(* CoDeSys 2.3 export: FB_LAMP.EXP *)

(* POU FBs/FB_Lamp, ST *)
(*
 TODO: REACTION
*)
FUNCTION_BLOCK FB_Lamp
VAR_INPUT
	ON_OFF: BOOL;   (* on/off on pulse, ignored if FORCE = TRUE *)
	ON: BOOL;   (* on on pulse, ignored if FORCE = TRUE *)
	OFF: BOOL;   (* off on pulse, ignored if FORCE = TRUE *)
	PT: TIME := t#30s;   (* auto-off aka on-time; see also: expandPT *)
	OFF_BLOCK_ON: TIME := t#15s;   (* after off block ON for the time specified *)
	REACTION: TIME := t#600ms;   (* TODO: do not change state right after statechange *)
	FORCE: BOOL;   (* if true, force output on/off, depending on FORCE_ON;
			  during FORCE, IN is ignored
			  during FORCE, PT is expanded if Q = TRUE *)
	FORCE_ON: BOOL;   (* if false and FORCE, then force off *)
	ROOM: STRING;
	LOCATION: STRING;
END_VAR
VAR_OUTPUT RETAIN PERSISTENT
	usageTime: TIME := t#0ms;
	usageDays: UINT := 0;
	usageCounterSwitchOn: UDINT := 0;
END_VAR
VAR_OUTPUT
	Q: BOOL;   (* lamp on / off *)
END_VAR
VAR
	viText: STRING; (* ro by visualisation *)
	viOnTimer: TIME; (* ro by visualisation *)
	viOffTimer: TIME; (* ro by visualisation *)
	viOnOff: BOOL; (* wo by visualisation *)
	onTimer: TOF;
	offTimer: TOF;
	onTrigger: R_TRIG;
	onOffTrigger: R_TRIG;
	offTrigger: R_TRIG;
	forceOnTrigger: R_TRIG;
	forceOffTrigger: F_TRIG;
	forceOnTime: TIME;
	startOpTrigger: R_TRIG;
	stopOpTrigger: F_TRIG;
	opTimetracker: TIME;
	now: TIME;
	extendPT: TIME;   (* added to onTimer.PT *)
END_VAR
VAR CONSTANT
	MAX_TIME: TIME := T#71582m47s295ms;
END_VAR
viText := CONCAT(ROOM, '$N');
viText := CONCAT(viText, LOCATION);
(* viOnTimer and viOffTimer are set later *)

now := TIME();

forceOnTrigger(CLK := FORCE);
forceOffTrigger(CLK := FORCE);
IF forceOnTrigger.Q AND onTimer.Q THEN
	forceOnTime := now;
ELSIF forceOffTrigger.Q AND onTimer.Q THEN
	IF (now < forceOnTime) THEN
		(* overflow *)
		extendPT := MAX_TIME - forceOnTime + now;
	ELSE
		extendPT := now - forceOnTime;
	END_IF
	onTimer.PT := onTimer.PT + extendPT;
END_IF

IF FORCE THEN
	Q := FORCE_ON;
ELSE (* NOT FORCE *)
	onTrigger(CLK := ON);
	onOffTrigger(CLK := ON_OFF XOR viOnOff);
	offTrigger(CLK := OFF);
	IF (onTrigger.Q OR onOffTrigger.Q) AND NOT onTimer.Q THEN   (* on or on/off pulse and onTimer = off *)
		IF onTrigger.Q AND offTimer.Q THEN
			(* ignore on while offTimer.Q is TRUE *)
			;
		ELSE
			(* turn on lamp and onTimer, reset offTimer *)
			onTimer(IN := TRUE, PT := PT);
			offTimer(IN := FALSE, PT := OFF_BLOCK_ON);
		END_IF
	ELSIF (offTrigger.Q OR onOffTrigger.Q) AND onTimer.Q THEN   (* off or on/off pulse and onTimer = on *)
		(* turn off timer / lamp *)
		onTimer(IN := FALSE, PT := t#0s);
		extendPT := t#0ms;
		offTimer(IN := TRUE, PT := OFF_BLOCK_ON);
	ELSIF onTrigger.Q AND onTimer.Q THEN   (* on pulse and onTimer = on *)
		(* reset PT *)
		onTimer(IN := TRUE, PT := PT);
 	ELSIF onTimer.Q THEN   (* no on/off pulse but timer is on *)
		onTimer(IN := FALSE);
	ELSIF offTimer.Q THEN
		offTimer(IN := FALSE);
	END_IF
	Q := onTimer.Q;
END_IF (* NOT FORCE *)

IF onTimer.ET = onTimer.PT THEN
	(* we do not want to see 0, when the onTimer is finished *)
	(* instead, display PT *)
	viOnTimer := PT;
ELSE
	viOnTimer := onTimer.PT - onTimer.ET;
END_IF
IF offTimer.ET = offTimer.PT THEN
	(* we do not want to see 0, when the offTimer is finished *)
	(* instead, display PT *)
	viOffTimer := OFF_BLOCK_ON;
ELSE
	viOffTimer := offTimer.PT - offTimer.ET;
END_IF

(*****************************)
(* record the operation time *)

startOpTrigger(CLK := Q);
stopOpTrigger(CLK := Q);
IF startOpTrigger.Q THEN
	usageCounterSwitchOn := usageCounterSwitchOn + 1;
	opTimetracker := now;
END_IF
IF Q AND (now < opTimetracker) THEN   (* overflow *)
	usageTime := usageTime + (MAX_TIME - opTimetracker);
	opTimetracker := t#0ms;
END_IF
IF stopOpTrigger.Q THEN
	usageTime := usageTime + (now - opTimetracker);
END_IF
IF Q AND ((now - opTimetracker) > t#1s) THEN
	usageTime := usageTime + (now - opTimetracker);
	opTimetracker := now;
END_IF
IF (Q OR stopOpTrigger.Q) AND (usageTime > t#1d) THEN
	usageDays := usageDays + 1;
	usageTime := usageTime - t#1d;
END_IF
END_FUNCTION_BLOCK
